KUKA KRL program: mo_seitlichZehn.src, mo_seitlichZehn.dat

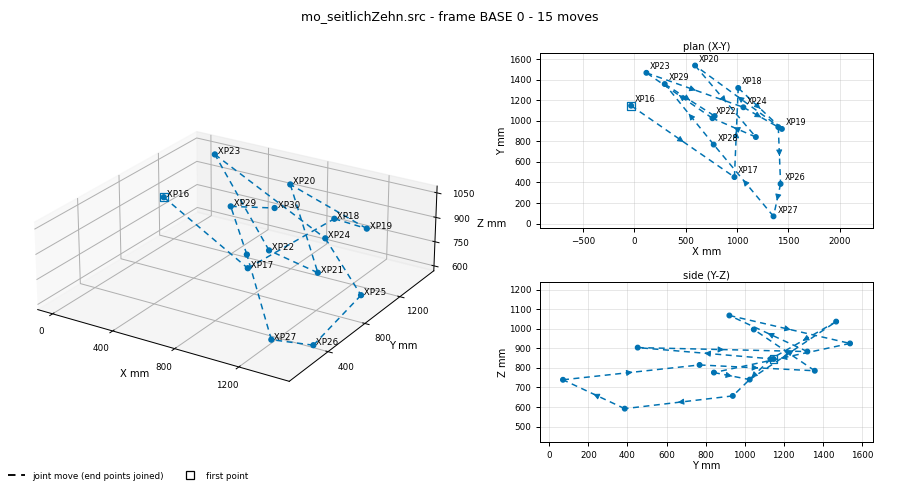
[picture p0: tool path of mo_seitlichZehn.src in frame BASE 0, 15 of 17 moves have a stored position in this frame; points joined in program order, loops and branches not executed]
--- mo_seitlichZehn.src ---
&ACCESS RVP
&REL 15
&PARAM EDITMASK = *
&PARAM TEMPLATE = C:\KRC\Roboter\Template\vorgabe
DEF mo_seitlichGewicht( )
;FOLD INI;%{PE}
  ;FOLD BASISTECH INI
    GLOBAL INTERRUPT DECL 3 WHEN $STOPMESS==TRUE DO IR_STOPM ( )
    INTERRUPT ON 3
    BAS (#INITMOV,0 )
  ;ENDFOLD (BASISTECH INI)
  ;FOLD USER INI
    ;Make your modifications here

  ;ENDFOLD (USER INI)
;ENDFOLD (INI)

FOR K=1 TO 200 STEP 1


;FOLD PTP HOME Vel=10 % DEFAULT;%{PE}%R 8.3.40,%MKUKATPBASIS,%CMOVE,%VPTP,%P 1:PTP, 2:HOME, 3:, 5:10, 7:DEFAULT
$BWDSTART=FALSE
PDAT_ACT=PDEFAULT
FDAT_ACT=FHOME
BAS(#PTP_PARAMS,10)
$H_POS=XHOME
PTP XHOME
;ENDFOLD

WAIT FOR IS_KEY_PRESSED(12)

;FOLD PTP P16 Vel=30 % PDAT16 Tool[11]:jan_ba Base[0];%{PE}%R 8.3.40,%MKUKATPBASIS,%CMOVE,%VPTP,%P 1:PTP, 2:P16, 3:, 5:30, 7:PDAT16
$BWDSTART=FALSE
PDAT_ACT=PPDAT16
FDAT_ACT=FP16
BAS(#PTP_PARAMS,30)
PTP XP16
;ENDFOLD

WAIT FOR IS_KEY_PRESSED(12)

;FOLD PTP P17 Vel=30 % PDAT17 Tool[11]:jan_ba Base[0];%{PE}%R 8.3.40,%MKUKATPBASIS,%CMOVE,%VPTP,%P 1:PTP, 2:P17, 3:, 5:30, 7:PDAT17
$BWDSTART=FALSE
PDAT_ACT=PPDAT17
FDAT_ACT=FP17
BAS(#PTP_PARAMS,30)
PTP XP17
;ENDFOLD

WAIT FOR IS_KEY_PRESSED(12)

;FOLD PTP P18 Vel=30 % PDAT18 Tool[11]:jan_ba Base[0];%{PE}%R 8.3.40,%MKUKATPBASIS,%CMOVE,%VPTP,%P 1:PTP, 2:P18, 3:, 5:30, 7:PDAT18
$BWDSTART=FALSE
PDAT_ACT=PPDAT18
FDAT_ACT=FP18
BAS(#PTP_PARAMS,30)
PTP XP18
;ENDFOLD

WAIT FOR IS_KEY_PRESSED(12)

;FOLD PTP P19 Vel=30 % PDAT19 Tool[11]:jan_ba Base[0];%{PE}%R 8.3.40,%MKUKATPBASIS,%CMOVE,%VPTP,%P 1:PTP, 2:P19, 3:, 5:30, 7:PDAT19
$BWDSTART=FALSE
PDAT_ACT=PPDAT19
FDAT_ACT=FP19
BAS(#PTP_PARAMS,30)
PTP XP19
;ENDFOLD

WAIT FOR IS_KEY_PRESSED(12)

;FOLD PTP P20 Vel=30 % PDAT20 Tool[11]:jan_ba Base[0];%{PE}%R 8.3.40,%MKUKATPBASIS,%CMOVE,%VPTP,%P 1:PTP, 2:P20, 3:, 5:30, 7:PDAT20
$BWDSTART=FALSE
PDAT_ACT=PPDAT20
FDAT_ACT=FP20
BAS(#PTP_PARAMS,30)
PTP XP20
;ENDFOLD

WAIT FOR IS_KEY_PRESSED(12)

;FOLD PTP P21 Vel=30 % PDAT21 Tool[11]:jan_ba Base[0];%{PE}%R 8.3.40,%MKUKATPBASIS,%CMOVE,%VPTP,%P 1:PTP, 2:P21, 3:, 5:30, 7:PDAT21
$BWDSTART=FALSE
PDAT_ACT=PPDAT21
FDAT_ACT=FP21
BAS(#PTP_PARAMS,30)
PTP XP21
;ENDFOLD

WAIT FOR IS_KEY_PRESSED(12)

;FOLD PTP P22 Vel=30 % PDAT22 Tool[11]:jan_ba Base[0];%{PE}%R 8.3.40,%MKUKATPBASIS,%CMOVE,%VPTP,%P 1:PTP, 2:P22, 3:, 5:30, 7:PDAT22
$BWDSTART=FALSE
PDAT_ACT=PPDAT22
FDAT_ACT=FP22
BAS(#PTP_PARAMS,30)
PTP XP22
;ENDFOLD

WAIT FOR IS_KEY_PRESSED(12)

;FOLD PTP P23 Vel=30 % PDAT23 Tool[11]:jan_ba Base[0];%{PE}%R 8.3.40,%MKUKATPBASIS,%CMOVE,%VPTP,%P 1:PTP, 2:P23, 3:, 5:30, 7:PDAT23
$BWDSTART=FALSE
PDAT_ACT=PPDAT23
FDAT_ACT=FP23
BAS(#PTP_PARAMS,30)
PTP XP23
;ENDFOLD

WAIT FOR IS_KEY_PRESSED(12)

;FOLD PTP P24 Vel=30 % PDAT24 Tool[11]:jan_ba Base[0];%{PE}%R 8.3.40,%MKUKATPBASIS,%CMOVE,%VPTP,%P 1:PTP, 2:P24, 3:, 5:30, 7:PDAT24
$BWDSTART=FALSE
PDAT_ACT=PPDAT24
FDAT_ACT=FP24
BAS(#PTP_PARAMS,30)
PTP XP24
;ENDFOLD

WAIT FOR IS_KEY_PRESSED(12)

;FOLD PTP P25 Vel=30 % PDAT25 Tool[11]:jan_ba Base[0];%{PE}%R 8.3.40,%MKUKATPBASIS,%CMOVE,%VPTP,%P 1:PTP, 2:P25, 3:, 5:30, 7:PDAT25
$BWDSTART=FALSE
PDAT_ACT=PPDAT25
FDAT_ACT=FP25
BAS(#PTP_PARAMS,30)
PTP XP25
;ENDFOLD

WAIT FOR IS_KEY_PRESSED(12)

;FOLD PTP P26 Vel=30 % PDAT26 Tool[11]:jan_ba Base[0];%{PE}%R 8.3.40,%MKUKATPBASIS,%CMOVE,%VPTP,%P 1:PTP, 2:P26, 3:, 5:30, 7:PDAT26
$BWDSTART=FALSE
PDAT_ACT=PPDAT26
FDAT_ACT=FP26
BAS(#PTP_PARAMS,30)
PTP XP26
;ENDFOLD

WAIT FOR IS_KEY_PRESSED(12)

;FOLD PTP P27 Vel=30 % PDAT27 Tool[11]:jan_ba Base[0];%{PE}%R 8.3.40,%MKUKATPBASIS,%CMOVE,%VPTP,%P 1:PTP, 2:P27, 3:, 5:30, 7:PDAT27
$BWDSTART=FALSE
PDAT_ACT=PPDAT27
FDAT_ACT=FP27
BAS(#PTP_PARAMS,30)
PTP XP27
;ENDFOLD

WAIT FOR IS_KEY_PRESSED(12)

;FOLD PTP P28 Vel=30 % PDAT28 Tool[11]:jan_ba Base[0];%{PE}%R 8.3.40,%MKUKATPBASIS,%CMOVE,%VPTP,%P 1:PTP, 2:P28, 3:, 5:30, 7:PDAT28
$BWDSTART=FALSE
PDAT_ACT=PPDAT28
FDAT_ACT=FP28
BAS(#PTP_PARAMS,30)
PTP XP28
;ENDFOLD

WAIT FOR IS_KEY_PRESSED(12)

;FOLD PTP P29 Vel=30 % PDAT29 Tool[11]:jan_ba Base[0];%{PE}%R 8.3.40,%MKUKATPBASIS,%CMOVE,%VPTP,%P 1:PTP, 2:P29, 3:, 5:30, 7:PDAT29
$BWDSTART=FALSE
PDAT_ACT=PPDAT29
FDAT_ACT=FP29
BAS(#PTP_PARAMS,30)
PTP XP29
;ENDFOLD

WAIT FOR IS_KEY_PRESSED(12)

;FOLD PTP P30 Vel=30 % PDAT30 Tool[11]:jan_ba Base[0];%{PE}%R 8.3.40,%MKUKATPBASIS,%CMOVE,%VPTP,%P 1:PTP, 2:P30, 3:, 5:30, 7:PDAT30
$BWDSTART=FALSE
PDAT_ACT=PPDAT30
FDAT_ACT=FP30
BAS(#PTP_PARAMS,30)
PTP XP30
;ENDFOLD

WAIT FOR IS_KEY_PRESSED(12)

;FOLD PTP HOME Vel=10 % DEFAULT;%{PE}%R 8.3.40,%MKUKATPBASIS,%CMOVE,%VPTP,%P 1:PTP, 2:HOME, 3:, 5:10, 7:DEFAULT
$BWDSTART=FALSE
PDAT_ACT=PDEFAULT
FDAT_ACT=FHOME
BAS(#PTP_PARAMS,10)
$H_POS=XHOME
PTP XHOME
;ENDFOLD

ENDFOR

END

--- mo_seitlichZehn.dat ---
&ACCESS RVP
&REL 15
&PARAM EDITMASK = *
&PARAM TEMPLATE = C:\KRC\Roboter\Template\vorgabe
DEFDAT  mo_seitlichGewicht
;FOLD EXTERNAL DECLARATIONS;%{PE}%MKUKATPBASIS,%CEXT,%VCOMMON,%P
;FOLD BASISTECH EXT;%{PE}%MKUKATPBASIS,%CEXT,%VEXT,%P
EXT  BAS (BAS_COMMAND  :IN,REAL  :IN )
DECL INT SUCCESS
;ENDFOLD (BASISTECH EXT)
;FOLD USER EXT;%{E}%MKUKATPUSER,%CEXT,%VEXT,%P
;Make your modifications here

;ENDFOLD (USER EXT)
;ENDFOLD (EXTERNAL DECLARATIONS)
DECL BASIS_SUGG_T LAST_BASIS={POINT1[] "P30                     ",POINT2[] "P30                     ",CP_PARAMS[] "CPDAT0                  ",PTP_PARAMS[] "PDAT30                  ",CONT[] "                        ",CP_VEL[] "2.0                     ",PTP_VEL[] "30                      ",SYNC_PARAMS[] "SYNCDAT                 ",SPL_NAME[] "S0                      ",A_PARAMS[] "ADAT0                   "}
DECL E6POS XP1={X -32.0779190,Y 1147.59277,Z 845.808838,A -110.239220,B 80.7838287,C 143.338074,S 22,T 51,E1 0.00492157834,E2 20159.9980,E3 0.0,E4 0.0,E5 0.0,E6 0.0}
DECL FDAT FP1={TOOL_NO 11,BASE_NO 0,IPO_FRAME #BASE,POINT2[] " ",TQ_STATE FALSE}
DECL PDAT PPDAT1={VEL 100.000,ACC 50.0000,APO_DIST 100.000,APO_MODE #CDIS,GEAR_JERK 50.0000,EXAX_IGN 0}
DECL E6POS XP2={X 1114.71143,Y 493.978577,Z 884.471863,A -160.957901,B 66.4580612,C 96.9383621,S 22,T 51,E1 0.00497351913,E2 20160.0,E3 0.0,E4 0.0,E5 0.0,E6 0.0}
DECL FDAT FP2={TOOL_NO 11,BASE_NO 0,IPO_FRAME #BASE,POINT2[] " ",TQ_STATE FALSE}
DECL PDAT PPDAT2={VEL 100.000,ACC 50.0000,APO_DIST 100.000,APO_MODE #CDIS,GEAR_JERK 50.0000,EXAX_IGN 0}
DECL E6POS XP3={X 1029.70459,Y 880.823425,Z 1404.86865,A -44.4400787,B 54.3737068,C -107.996033,S 22,T 51,E1 0.00497351913,E2 20160.0,E3 0.0,E4 0.0,E5 0.0,E6 0.0}
DECL FDAT FP3={TOOL_NO 11,BASE_NO 0,IPO_FRAME #BASE,POINT2[] " ",TQ_STATE FALSE}
DECL PDAT PPDAT3={VEL 100.000,ACC 50.0000,APO_DIST 100.000,APO_MODE #CDIS,GEAR_JERK 50.0000,EXAX_IGN 0}
DECL E6POS XP4={X 1143.06104,Y 1312.88147,Z 778.726257,A -110.383789,B 27.8682251,C -167.688232,S 18,T 3,E1 0.00497351913,E2 20160.0,E3 0.0,E4 0.0,E5 0.0,E6 0.0}
DECL FDAT FP4={TOOL_NO 11,BASE_NO 0,IPO_FRAME #BASE,POINT2[] " ",TQ_STATE FALSE}
DECL PDAT PPDAT4={VEL 100.000,ACC 50.0000,APO_DIST 100.000,APO_MODE #CDIS,GEAR_JERK 50.0000,EXAX_IGN 0}
DECL E6POS XP5={X 829.158447,Y 1604.10913,Z 1075.56653,A 158.441864,B 1.04213142,C 82.5205231,S 22,T 51,E1 0.00497351913,E2 20160.0,E3 0.0,E4 0.0,E5 0.0,E6 0.0}
DECL FDAT FP5={TOOL_NO 11,BASE_NO 0,IPO_FRAME #BASE,POINT2[] " ",TQ_STATE FALSE}
DECL PDAT PPDAT5={VEL 100.000,ACC 50.0000,APO_DIST 100.000,APO_MODE #CDIS,GEAR_JERK 50.0000,EXAX_IGN 0}
DECL E6POS XP6={X 854.191406,Y 1682.95190,Z 710.727539,A -106.355331,B 54.5122948,C 177.907654,S 22,T 51,E1 0.00497351913,E2 20160.0,E3 0.0,E4 0.0,E5 0.0,E6 0.0}
DECL FDAT FP6={TOOL_NO 11,BASE_NO 0,IPO_FRAME #BASE,POINT2[] " ",TQ_STATE FALSE}
DECL PDAT PPDAT6={VEL 100.000,ACC 50.0000,APO_DIST 100.000,APO_MODE #CDIS,GEAR_JERK 50.0000,EXAX_IGN 0}
DECL E6POS XP7={X 430.342529,Y 1926.08496,Z 864.580383,A -130.642166,B 64.7543182,C 157.692810,S 18,T 35,E1 0.00497351913,E2 20160.0,E3 0.0,E4 0.0,E5 0.0,E6 0.0}
DECL FDAT FP7={TOOL_NO 11,BASE_NO 0,IPO_FRAME #BASE,POINT2[] " ",TQ_STATE FALSE}
DECL PDAT PPDAT7={VEL 100.000,ACC 50.0000,APO_DIST 100.000,APO_MODE #CDIS,GEAR_JERK 50.0000,EXAX_IGN 0}
DECL E6POS XP8={X 276.902344,Y 1867.76904,Z 489.372284,A -160.351288,B 72.1188049,C 91.3736,S 18,T 35,E1 0.00497351913,E2 20160.0,E3 0.0,E4 0.0,E5 0.0,E6 0.0}
DECL FDAT FP8={TOOL_NO 11,BASE_NO 0,IPO_FRAME #BASE,POINT2[] " ",TQ_STATE FALSE}
DECL PDAT PPDAT8={VEL 100.000,ACC 50.0000,APO_DIST 100.000,APO_MODE #CDIS,GEAR_JERK 50.0000,EXAX_IGN 0}
DECL E6POS XP9={X 163.911804,Y 1351.15894,Z 655.545776,A 5.89288568,B 83.1484222,C -142.337936,S 18,T 35,E1 0.00497351913,E2 20160.0,E3 0.0,E4 0.0,E5 0.0,E6 0.0}
DECL FDAT FP9={TOOL_NO 11,BASE_NO 0,IPO_FRAME #BASE,POINT2[] " ",TQ_STATE FALSE}
DECL PDAT PPDAT9={VEL 100.000,ACC 50.0000,APO_DIST 100.000,APO_MODE #CDIS,GEAR_JERK 50.0000,EXAX_IGN 0}
DECL E6POS XP10={X 234.619431,Y 1275.68262,Z 681.751831,A -165.034714,B 22.9009,C 145.619919,S 18,T 35,E1 0.00497351913,E2 20160.0,E3 0.0,E4 0.0,E5 0.0,E6 0.0}
DECL FDAT FP10={TOOL_NO 11,BASE_NO 0,IPO_FRAME #BASE,POINT2[] " ",TQ_STATE FALSE}
DECL PDAT PPDAT10={VEL 100.000,ACC 50.0000,APO_DIST 100.000,APO_MODE #CDIS,GEAR_JERK 50.0000,EXAX_IGN 0}
DECL E6POS XP11={X 743.968,Y 959.536438,Z 920.631,A -134.732986,B 27.2720585,C 176.965302,S 22,T 51,E1 0.00497351913,E2 20160.0,E3 0.0,E4 0.0,E5 0.0,E6 0.0}
DECL FDAT FP11={TOOL_NO 11,BASE_NO 0,IPO_FRAME #BASE,POINT2[] " ",TQ_STATE FALSE}
DECL PDAT PPDAT11={VEL 100.000,ACC 50.0000,APO_DIST 100.000,APO_MODE #CDIS,GEAR_JERK 50.0000,EXAX_IGN 0}
DECL E6POS XP12={X 1013.13965,Y 565.329529,Z 778.797607,A -166.777634,B 65.3451767,C 123.284828,S 18,T 35,E1 0.00497351913,E2 20160.0,E3 0.0,E4 0.0,E5 0.0,E6 0.0}
DECL FDAT FP12={TOOL_NO 11,BASE_NO 0,IPO_FRAME #BASE,POINT2[] " ",TQ_STATE FALSE}
DECL PDAT PPDAT12={VEL 100.000,ACC 50.0000,APO_DIST 100.000,APO_MODE #CDIS,GEAR_JERK 50.0000,EXAX_IGN 0}
DECL E6POS XP13={X 1240.05823,Y 794.612915,Z 795.552490,A -136.986664,B 36.8687286,C 98.6252747,S 18,T 35,E1 0.00497351913,E2 20160.0,E3 0.0,E4 0.0,E5 0.0,E6 0.0}
DECL FDAT FP13={TOOL_NO 11,BASE_NO 0,IPO_FRAME #BASE,POINT2[] " ",TQ_STATE FALSE}
DECL PDAT PPDAT13={VEL 100.000,ACC 50.0000,APO_DIST 100.000,APO_MODE #CDIS,GEAR_JERK 50.0000,EXAX_IGN 0}
DECL E6POS XP14={X 1707.50085,Y 839.382629,Z 728.205872,A 107.462547,B 67.2460709,C 78.7145538,S 18,T 35,E1 0.00499581080,E2 20160.0,E3 0.0,E4 0.0,E5 0.0,E6 0.0}
DECL FDAT FP14={TOOL_NO 11,BASE_NO 0,IPO_FRAME #BASE,POINT2[] " ",TQ_STATE FALSE}
DECL PDAT PPDAT14={VEL 100.000,ACC 50.0000,APO_DIST 100.000,APO_MODE #CDIS,GEAR_JERK 50.0000,EXAX_IGN 0}
DECL E6POS XP15={X 127.119453,Y 1397.62366,Z 966.970276,A 29.0370808,B 72.7731247,C -80.1114655,S 18,T 35,E1 0.00499581080,E2 20160.0,E3 0.0,E4 0.0,E5 0.0,E6 0.0}
DECL FDAT FP15={TOOL_NO 11,BASE_NO 0,IPO_FRAME #BASE,POINT2[] " ",TQ_STATE FALSE}
DECL PDAT PPDAT15={VEL 100.000,ACC 50.0000,APO_DIST 100.000,APO_MODE #CDIS,GEAR_JERK 50.0000,EXAX_IGN 0}
DECL E6POS XP16={X -32.0779190,Y 1147.59277,Z 845.808838,A -110.239220,B 80.7838287,C 143.338074,S 22,T 51,E1 0.00492157834,E2 20159.9980,E3 0.0,E4 0.0,E5 0.0,E6 0.0}
DECL FDAT FP16={TOOL_NO 11,BASE_NO 0,IPO_FRAME #BASE,POINT2[] " ",TQ_STATE FALSE}
DECL PDAT PPDAT16={VEL 100.000,ACC 50.0000,APO_DIST 100.000,APO_MODE #CDIS,GEAR_JERK 50.0000,EXAX_IGN 0}
DECL E6POS XP17={X 974.307190,Y 452.404938,Z 904.120361,A -32.5194931,B 75.0684280,C -91.5796,S 22,T 19,E1 0.00492157834,E2 20159.9980,E3 0.0,E4 0.0,E5 0.0,E6 0.0}
DECL FDAT FP17={TOOL_NO 11,BASE_NO 0,IPO_FRAME #BASE,POINT2[] " ",TQ_STATE FALSE}
DECL PDAT PPDAT17={VEL 100.000,ACC 50.0000,APO_DIST 100.000,APO_MODE #CDIS,GEAR_JERK 50.0000,EXAX_IGN 0}
DECL E6POS XP18={X 1011.20044,Y 1320.68359,Z 883.862305,A -98.1202393,B 76.6139069,C -163.671539,S 22,T 51,E1 0.00492157834,E2 20159.9980,E3 0.0,E4 0.0,E5 0.0,E6 0.0}
DECL FDAT FP18={TOOL_NO 11,BASE_NO 0,IPO_FRAME #BASE,POINT2[] " ",TQ_STATE FALSE}
DECL PDAT PPDAT18={VEL 100.000,ACC 50.0000,APO_DIST 100.000,APO_MODE #CDIS,GEAR_JERK 50.0000,EXAX_IGN 0}
DECL E6POS XP19={X 1436.40320,Y 921.601563,Z 1068.45618,A 161.447540,B 58.8285522,C 135.093246,S 22,T 59,E1 0.00492157834,E2 20159.9980,E3 0.0,E4 0.0,E5 0.0,E6 0.0}
DECL FDAT FP19={TOOL_NO 11,BASE_NO 0,IPO_FRAME #BASE,POINT2[] " ",TQ_STATE FALSE}
DECL PDAT PPDAT19={VEL 100.000,ACC 50.0000,APO_DIST 100.000,APO_MODE #CDIS,GEAR_JERK 50.0000,EXAX_IGN 0}
DECL E6POS XP20={X 591.003906,Y 1539.06055,Z 925.462402,A -57.0219688,B 78.8618088,C -151.421188,S 22,T 51,E1 0.00492157834,E2 20159.9980,E3 0.0,E4 0.0,E5 0.0,E6 0.0}
DECL FDAT FP20={TOOL_NO 11,BASE_NO 0,IPO_FRAME #BASE,POINT2[] " ",TQ_STATE FALSE}
DECL PDAT PPDAT20={VEL 100.000,ACC 50.0000,APO_DIST 100.000,APO_MODE #CDIS,GEAR_JERK 50.0000,EXAX_IGN 0}
DECL E6POS XP21={X 1182.80457,Y 842.501587,Z 776.382080,A -177.724319,B 43.2824745,C 155.580276,S 22,T 51,E1 0.00492157834,E2 20159.9980,E3 0.0,E4 0.0,E5 0.0,E6 0.0}
DECL FDAT FP21={TOOL_NO 11,BASE_NO 0,IPO_FRAME #BASE,POINT2[] " ",TQ_STATE FALSE}
DECL PDAT PPDAT21={VEL 100.000,ACC 50.0000,APO_DIST 100.000,APO_MODE #CDIS,GEAR_JERK 50.0000,EXAX_IGN 0}
DECL E6POS XP22={X 759.970032,Y 1025.67102,Z 740.416077,A -174.991074,B 79.8193,C 149.673,S 22,T 59,E1 0.00492157834,E2 20159.9980,E3 0.0,E4 0.0,E5 0.0,E6 0.0}
DECL FDAT FP22={TOOL_NO 11,BASE_NO 0,IPO_FRAME #BASE,POINT2[] " ",TQ_STATE FALSE}
DECL PDAT PPDAT22={VEL 100.000,ACC 50.0000,APO_DIST 100.000,APO_MODE #CDIS,GEAR_JERK 50.0000,EXAX_IGN 0}
DECL E6POS XP23={X 116.778374,Y 1468.06128,Z 1037.21362,A -131.086502,B 76.2769089,C 133.188644,S 22,T 51,E1 0.00492157834,E2 20159.9980,E3 0.0,E4 0.0,E5 0.0,E6 0.0}
DECL FDAT FP23={TOOL_NO 11,BASE_NO 0,IPO_FRAME #BASE,POINT2[] " ",TQ_STATE FALSE}
DECL PDAT PPDAT23={VEL 100.000,ACC 50.0000,APO_DIST 100.000,APO_MODE #CDIS,GEAR_JERK 50.0000,EXAX_IGN 0}
DECL E6POS XP24={X 1061.38867,Y 1132.27332,Z 845.179382,A -115.800789,B 21.9125557,C -166.459106,S 18,T 35,E1 0.00492157834,E2 20159.9980,E3 0.0,E4 0.0,E5 0.0,E6 0.0}
DECL FDAT FP24={TOOL_NO 11,BASE_NO 0,IPO_FRAME #BASE,POINT2[] " ",TQ_STATE FALSE}
DECL PDAT PPDAT24={VEL 100.000,ACC 50.0000,APO_DIST 100.000,APO_MODE #CDIS,GEAR_JERK 50.0000,EXAX_IGN 0}
DECL E6POS XP25={X 1401.62952,Y 939.120056,Z 656.911316,A -121.845291,B 48.9283447,C -176.857452,S 22,T 51,E1 0.00492157834,E2 20159.9980,E3 0.0,E4 0.0,E5 0.0,E6 0.0}
DECL FDAT FP25={TOOL_NO 11,BASE_NO 0,IPO_FRAME #BASE,POINT2[] " ",TQ_STATE FALSE}
DECL PDAT PPDAT25={VEL 100.000,ACC 50.0000,APO_DIST 100.000,APO_MODE #CDIS,GEAR_JERK 50.0000,EXAX_IGN 0}
DECL E6POS XP26={X 1423.60474,Y 386.033386,Z 591.663147,A 154.883759,B 32.7368088,C 161.013840,S 22,T 59,E1 0.00492157834,E2 20159.9980,E3 0.0,E4 0.0,E5 0.0,E6 0.0}
DECL FDAT FP26={TOOL_NO 11,BASE_NO 0,IPO_FRAME #BASE,POINT2[] " ",TQ_STATE FALSE}
DECL PDAT PPDAT26={VEL 100.000,ACC 50.0000,APO_DIST 100.000,APO_MODE #CDIS,GEAR_JERK 50.0000,EXAX_IGN 0}
DECL E6POS XP27={X 1354.82349,Y 69.9751892,Z 739.387573,A 172.077728,B 57.6340408,C -179.014572,S 22,T 27,E1 0.00492157834,E2 20159.9980,E3 0.0,E4 0.0,E5 0.0,E6 0.0}
DECL FDAT FP27={TOOL_NO 11,BASE_NO 0,IPO_FRAME #BASE,POINT2[] " ",TQ_STATE FALSE}
DECL PDAT PPDAT27={VEL 100.000,ACC 50.0000,APO_DIST 100.000,APO_MODE #CDIS,GEAR_JERK 50.0000,EXAX_IGN 0}
DECL E6POS XP28={X 772.071167,Y 769.101,Z 815.324463,A -99.7352448,B 81.9052048,C -166.371429,S 22,T 51,E1 0.00492157834,E2 20159.9980,E3 0.0,E4 0.0,E5 0.0,E6 0.0}
DECL FDAT FP28={TOOL_NO 11,BASE_NO 0,IPO_FRAME #BASE,POINT2[] " ",TQ_STATE FALSE}
DECL PDAT PPDAT28={VEL 100.000,ACC 50.0000,APO_DIST 100.000,APO_MODE #CDIS,GEAR_JERK 50.0000,EXAX_IGN 0}
DECL E6POS XP29={X 295.388824,Y 1358.67383,Z 785.581604,A -74.9102859,B 77.9381104,C 172.747513,S 22,T 51,E1 0.00492157834,E2 20159.9980,E3 0.0,E4 0.0,E5 0.0,E6 0.0}
DECL FDAT FP29={TOOL_NO 11,BASE_NO 0,IPO_FRAME #BASE,POINT2[] " ",TQ_STATE FALSE}
DECL PDAT PPDAT29={VEL 100.000,ACC 50.0000,APO_DIST 100.000,APO_MODE #CDIS,GEAR_JERK 50.0000,EXAX_IGN 0}
DECL E6POS XP30={X 781.739746,Y 1046.73450,Z 996.689148,A -73.5318146,B 89.2929764,C -132.984909,S 22,T 51,E1 0.00492157834,E2 20159.9980,E3 0.0,E4 0.0,E5 0.0,E6 0.0}
DECL FDAT FP30={TOOL_NO 11,BASE_NO 0,IPO_FRAME #BASE,POINT2[] " ",TQ_STATE FALSE}
DECL PDAT PPDAT30={VEL 100.000,ACC 50.0000,APO_DIST 100.000,APO_MODE #CDIS,GEAR_JERK 50.0000,EXAX_IGN 0}
ENDDAT
